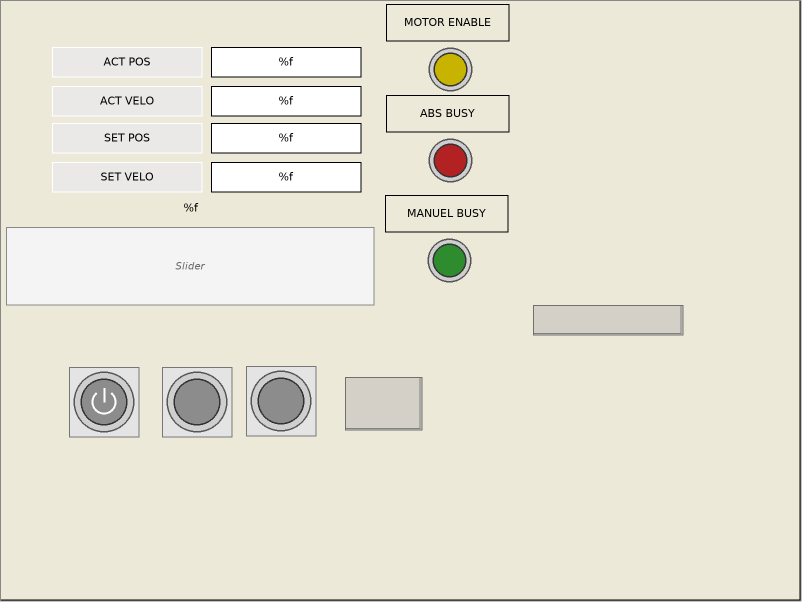
VISUALIZATION TC_SERVO1  // 802x602
    Rectangle (0,0 800x600)
    Rectangle (52,47 150x30), "ACT POS"
    Rectangle (211,47 150x30), "%f", text variable: Axis1.NcToPlc.ActPos
    Rectangle (52,86 150x30), "ACT VELO"
    Rectangle (211,86 150x30), "%f", text variable: Axis1.NcToPlc.ActVelo
    Rectangle (52,123 150x30), "SET POS"
    Rectangle (211,123 150x30), "%f", text variable: MAIN.fPos1
        OnMouseClick: write the text variable via VisuDialogs.Numpad
    Rectangle (52,162 150x30), "SET VELO"
    Rectangle (211,162 150x30), "%f", text variable: MAIN.fVelocity1
        OnMouseClick: write the text variable via VisuDialogs.Numpad
    Slider (6,227 368x78), variable: MAIN.fOverride1, scale 0..100
    Rectangle (160,194 62x28), "%f", text variable: MAIN.fOverride1
    PowerSwitch (69,367 70x70), variable: MAIN.bEnable1, behaviour: TOGGLE, style: Switch-PowerSwitch-Gray
    PushSwitch (162,367 70x70), variable: MAIN.bManuelBw1, behaviour: TOGGLE, style: Switch-PushSwitch-Gray
    PushSwitch (246,366 70x70), variable: MAIN.bManuelFw1, behaviour: TOGGLE, style: Switch-PushSwitch-Gray
    Button (345,377 77x53)
        tap MAIN.bMoveAbs1
    Lamp1 (424,44 53x51), variable: MAIN.bEnabled1, style: Lamp-Lamp1-Yellow
    Rectangle (386,4 123x37), "MOTOR ENABLE"
    Lamp1 (424,135 53x51), variable: MAIN.bMoveAbsBusy1, style: Lamp-Lamp1-Red
    Rectangle (386,95 123x37), "ABS BUSY"
    Lamp1 (423,235 53x51), variable: MAIN.bJogBusy1, style: Lamp-Lamp1-Green
    Rectangle (385,195 123x37), "MANUEL BUSY"
    Button (533,305 150x30)
END_VISUALIZATION

(* stored: Version 1.1.0.1, ProductVersion 3.1.4022.12
   Visu TC_SERVO1: Id {d7b99584-e02e-4252-81bf-9e13be0dc5ef} *)
